Yaskawa INFORM job: ROVI_CAPTURE.JBI

/JOB
//NAME ROVI_CAPTURE
///FOLDERNAME ROVI
//POS
///NPOS 0,0,0,0,0,0
//INST
///DATE 2019/12/05 15:04
///ATTR SC,RW
///GROUP1 RB1
///LVARS 0,2,0,0,0,0,0,0
NOP
SET LI000 I092
SET LI001 0
*CAPTURE
SET B080 1
WAIT B080=255
INC LI001
IFTHENEXP I080<>0
	 RET I080 IF LI001>=LI000
	 TIMER T=0.500
	 JUMP *CAPTURE
ENDIF
RET I080
END
